PROGRAM MAIN
VAR
	X1: BOOL;
	X2: BOOL;
	Y1: BOOL;
END_VAR

Main.ACT();

ACTION ACT:
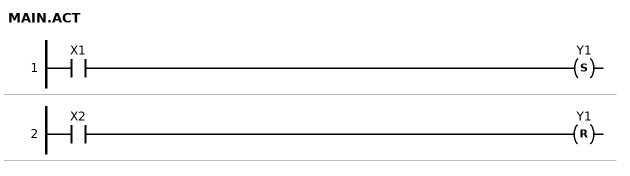
// NETWORK 1
Y1 S= X1;

// NETWORK 2
Y1 R= X2;
END_ACTION

END_PROGRAM

(* stored: Version 1.1.0.1, ProductVersion 3.1.4024.12
   POU MAIN: Id {302b8438-89a6-48af-b822-633e53125890}, SpecialFunc None
   Action ACT: Id {d806b113-d1eb-4171-9bbc-8398c53b359e} *)
